PROGRAM testSlitApp
VAR
    southBlade_ID : UINT := 2;
    northBlade_ID : UINT := 1;   
    VG_ID : UINT := 3;
    VC_ID : UINT := 4;
    bEnable : BOOL :=FALSE;
    
    
    
    fGapSizePosition: LREAL;
    iGapSizePosition AT %Q*: UDINT := 0;
    fGapCentrePosition: LREAL;
    iGapCentrePosition AT %Q*: UDINT := 0;
    fEncoderScaling : LREAL := 10000;
    
    northSpGenEnable : MC_ExtSetPointGenEnable;
    northSpGenDisable : MC_ExtSetPointGenDisable;
    southSpGenEnable : MC_ExtSetPointGenEnable;
    southSpGenDisable : MC_ExtSetPointGenDisable;
    
    vgSpGenEnable : MC_ExtSetPointGenEnable;
    vgSpGenDisable : MC_ExtSetPointGenDisable;
    vcSpGenEnable : MC_ExtSetPointGenEnable;
    vcSpGenDisable : MC_ExtSetPointGenDisable;
    
    fNorthSp : LREAL;
    fSouthSp : LREAL;
    fVgSp : LREAL;
    fVcSp : LREAL;
    fNorthVelSp : LREAL;
    fSouthVelSp : LREAL;
    fVgVelSp:LREAL;
    fVcVelSp : LREAL;
    
    northDir : DINT;
    southDir : DINT;
    vgDir : DINT;
    vcDir : DINT;
    
    
    lastCycleSP_North : LREAL;
    lastCycleSP_South : LREAL;
    lastCycleSP_VG : LREAL;
    lastCycleSP_VC : LREAL;
    
    iState : UINT := 0;

END_VAR

actVirtualAxisPositions();
//IF bEnable THEN

GVL.astAxes[northBlade_ID].stControl.bEnable:=TRUE;
GVL.astAxes[southBlade_ID].stControl.bEnable:=TRUE;
GVL.astAxes[VG_ID].stControl.bEnable:=TRUE;
GVL.astAxes[VC_ID].stControl.bEnable:=TRUE;
GVL.astAxes[5].stControl.bEnable:=TRUE;
GVL.astAxes[6].stControl.bEnable:=TRUE;
GVL.astAxes[VG_ID].stInputs.bLimitBwd := TRUE;
GVL.astAxes[VG_ID].stInputs.bLimitFwd := TRUE;
GVL.astAxes[VC_ID].stInputs.bLimitBwd := TRUE;
GVL.astAxes[VC_ID].stInputs.bLimitFwd := TRUE;
GVL.astAxes[5].stInputs.bLimitBwd := TRUE;
GVL.astAxes[5].stInputs.bLimitFwd := TRUE;
GVL.astAxes[6].stInputs.bLimitBwd := TRUE;
GVL.astAxes[6].stInputs.bLimitFwd := TRUE;

northSpGenEnable(Axis:= GVL.astAxes[northBlade_ID].Axis);
northSpGenEnable.Execute:=FALSE;
southSpGenEnable(Axis:=GVL.astAxes[southBlade_ID].Axis);
southSpGenEnable.Execute:=FALSE;
northSpGenDisable(Axis:= GVL.astAxes[northBlade_ID].Axis);
northSpGenDisable.Execute:=FALSE;
southSpGenDisable(Axis:=GVL.astAxes[southBlade_ID].Axis);
southSpGenDisable.Execute:=FALSE;

vgSpGenEnable(Axis:= GVL.astAxes[3].Axis);
vgSpGenEnable.Execute:=FALSE;
vcSpGenEnable(Axis:=GVL.astAxes[4].Axis);
vcSpGenEnable.Execute:=FALSE;
vgSpGenDisable(Axis:= GVL.astAxes[3].Axis);
vgSpGenDisable.Execute:=FALSE;
vcSpGenDisable(Axis:=GVL.astAxes[4].Axis);
vcSpGenDisable.Execute:=FALSE;

fNorthSp := GVL.astAxes[VC_ID].Axis.NcToPlc.SetPos + (GVL.astAxes[VG_ID].Axis.NcToPlc.SetPos/2);
fSouthSp := GVL.astAxes[VC_ID].Axis.NcToPlc.SetPos - (GVL.astAxes[VG_ID].Axis.NcToPlc.SetPos/2);
fNorthVelSp := GVL.astAxes[VC_ID].Axis.NcToPlc.SetVelo +(GVL.astAxes[VG_ID].Axis.NcToPlc.SetVelo/2) + GVL.astAxes[5].Axis.NcToPlc.SetVelo;
fSouthVelSp := GVL.astAxes[VC_ID].Axis.NcToPlc.SetVelo -(GVL.astAxes[VG_ID].Axis.NcToPlc.SetVelo/2) + GVL.astAxes[6].Axis.NcToPlc.SetVelo;
IF fNorthVelSp>0 THEN
    northDir := 1;
ELSIF fNorthVelSp<0 THEN
    northDir:=-1;
ELSE 
    northDir:=0;
END_IF
IF fSouthVelSp>0 THEN
    SouthDir := 1;
ELSIF fSouthVelSp<0 THEN
    SouthDir:=-1;
ELSE 
    SouthDir:=0;
END_IF

fVgVelSp := GVL.astAxes[1].Axis.NcToPlc.SetVelo - GVL.astAxes[2].Axis.NcToPlc.SetVelo;
fVcVelSp := GVL.astAxes[1].Axis.NcToPlc.SetVelo + GVL.astAxes[2].Axis.NcToPlc.SetVelo;

IF fVgVelSp>0 THEN
    vgDir := 1;
ELSIF fVgVelSp<0 THEN
    vgDir:=-1;
ELSE 
    vgDir:=0;
END_IF
IF fVcVelSp>0 THEN
    vcDir := 1;
ELSIF fVcVelSp<0 THEN
    vcDir:=-1;
ELSE 
    vcDir:=0;
END_IF


fVgSp := GVL.astAxes[northBlade_ID].Axis.NcToPlc.SetPos - GVL.astAxes[southBlade_ID].Axis.NcToPlc.SetPos;
fVcSp := (GVL.astAxes[northBlade_ID].Axis.NcToPlc.SetPos + GVL.astAxes[southBlade_ID].Axis.NcToPlc.SetPos) / 2;



//IF northSpGenEnable.Enabled OR southSpGenEnable THEN
    //
//END_IF

    CASE istate OF
        0:
            IF GVL.astAxes[VG_ID].stStatus.bMoving OR GVL.astAxes[VC_ID].stStatus.bMoving THEN
                iState:=1;
			END_IF
            IF GVL.astAxes[1].stStatus.bMoving OR GVL.astAxes[2].stStatus.bMoving THEN
                iState:=10;
            END_IF
            
        1:
            northSpGenEnable.Execute:=TRUE;
            southSpGenEnable.Execute:=TRUE;
            iState:=2;
        2:
            IF NOT(GVL.astAxes[VG_ID].stStatus.bMoving OR GVL.astAxes[VC_ID].stStatus.bMoving) THEN
                iState:=3;
			END_IF
        3:
            northSpGenDisable.Execute:=TRUE;
            southSpGenDisable.Execute:=TRUE;
            iState:=0;
            
        10:
            vgSpGenEnable.Execute :=TRUE;
            vcSpGenEnable.Execute:=TRUE;
            iState:=11;
        11:
            IF NOT(GVL.astAxes[1].stStatus.bMoving OR GVL.astAxes[2].stStatus.bMoving) THEN
                iState:=12;
			END_IF
        12:
            vgSpGenDisable.Execute :=TRUE;
            vcSpGenDisable.Execute:=TRUE;
            iState:=0;
    
	END_CASE
(*IF (GVL.astAxes[VG_ID].stStatus.bMoving OR GVL.astAxes[VC_ID].stStatus.bMoving) AND NOT(vgSpGenEnable.Enabled OR vcSpGenEnable.Enabled) THEN
    northSpGenEnable.Execute:=TRUE;
    southSpGenEnable.Execute:=TRUE;
END_IF
IF NOT(GVL.astAxes[VG_ID].stStatus.bMoving) AND NOT(GVL.astAxes[VC_ID].stStatus.bMoving) THEN
    northSpGenDisable.Execute:=TRUE;
    southSpGenDisable.Execute:=TRUE;
END_IF
IF GVL.astAxes[1].stStatus.bMoving OR GVL.astAxes[2].stStatus.bMoving AND NOT(northSpGenEnable.Enabled OR southSpGenEnable.Enabled) AND NOT(northSpGenEnable.Execute)  THEN
    vgSpGenEnable.Execute :=TRUE;
    vcSpGenEnable.Execute:=TRUE;
END_IF
IF NOT(GVL.astAxes[1].stStatus.bMoving) AND NOT(GVL.astAxes[2].stStatus.bMoving) THEN
    vgSpGenDisable.Execute :=TRUE;
    vcSpGenDisable.Execute:=TRUE;
END_IF*)




MC_ExtSetPointGenFeed(Axis:= GVL.astAxes[northBlade_ID].Axis, Position:= fNorthSp, Velocity:=fNorthVelSp, Acceleration:=0,Direction:=northDir);
MC_ExtSetPointGenFeed(Axis:= GVL.astAxes[southBlade_ID].Axis, Position:= fSouthSp, Velocity:=fSouthVelSp, Acceleration:=0,Direction:=southDir);
MC_ExtSetPointGenFeed(Axis:= GVL.astAxes[3].Axis, Position:= fVgSp, Velocity:=fVgVelSp, Acceleration:=0,Direction:=vgDir);
MC_ExtSetPointGenFeed(Axis:= GVL.astAxes[4].Axis, Position:= fVcSp, Velocity:=fVcVelSp, Acceleration:=0,Direction:=vcDir);
 



lastCycleSP_North := GVL.astAxes[1].Axis.NcToPlc.SetPos;
lastCycleSP_South := GVL.astAxes[2].Axis.NcToPlc.SetPos;
lastCycleSP_VG := GVL.astAxes[3].Axis.NcToPlc.SetPos;
lastCycleSP_VC := GVL.astAxes[4].Axis.NcToPlc.SetPos;







//END_IF

ACTION actVirtualAxisPositions:
(*Calculate virtual axis positions and convert to UDINT.
Conversion to UDINT is prohibited if it would exceed UDINT max value of 4,294,967,295.
If this is not done, it can cause overflow when connected to the encoder input and hard-crash the PLC which will only recover with a power cycle.
To preserve decimal position data of the LREAL (i.e. anything <1mm) it is necessary to scale the value before converting to UDINT.
This can be reversed with the correct scaling at the NC encoder level.
*)
fGapSizePosition := GVL.astAxes[northBlade_ID].stStatus.fActPosition - GVL.astAxes[southBlade_ID].stStatus.fActPosition;
fGapCentrePosition := (GVL.astAxes[northBlade_ID].stStatus.fActPosition + GVL.astAxes[southBlade_ID].stStatus.fActPosition) / 2;


    IF ABS(fGapSizePosition) < 100000 THEN
        iGapSizePosition := LREAL_TO_UDINT(fGapSizePosition*fEncoderScaling);
    END_IF
    IF ABS(fGapCentrePosition) < 100000 THEN
        iGapCentrePosition := LREAL_TO_UDINT(fGapCentrePosition*fEncoderScaling);
    END_IF
END_ACTION

END_PROGRAM

(* stored: Version 1.1.0.1, ProductVersion 3.1.4024.5
   POU testSlitApp: Id {02dd3d5e-b93a-47d0-a30a-b16df70390e6}, SpecialFunc None
   Action actVirtualAxisPositions: Id {84408ed0-12a9-4a20-9ee2-393320dd5a43} *)
